(* Logix 5000 project; controller DUNEW2PLC1 vendor 1 type 14 code 221 rev 33.11; software revision 33.00; part 2 of 7 *)
(* tags used below, declared in another part *)
   AbortActive : BOOL;
   BOOLS : BOOL[1024];
   CheckCurSeg : BOOL;
   CheckNextSeg : BOOL;
   CmdA_Accel : REAL;
   CmdA_CircleType : DINT;
   CmdA_Decel : REAL;
   CmdA_Direction : DINT;
   CmdA_JerkAccel : REAL;
   CmdA_JerkDecel : REAL;
   CmdA_SegType : DINT;
   CmdA_Speed : REAL;
   CmdA_TermType : SINT;
   CmdA_ViaCenter : REAL[2];
   CmdA_XY : REAL[2];
   CmdB_Accel : REAL;
   CmdB_CircleType : DINT;
   CmdB_Decel : REAL;
   CmdB_Direction : DINT;
   CmdB_JerkAccel : REAL;
   CmdB_JerkDecel : REAL;
   CmdB_SegType : DINT;
   CmdB_Speed : REAL;
   CmdB_TermType : SINT;
   CmdB_ViaCenter : REAL[2];
   CmdB_XY : REAL[2];
   CmdTolerance : DINT;
   CurSeg : MotionSeg;
   DINTS : DINT[1024];
   EnqueueReq : BOOL;
   FaultCode : DINT;
   idx_0 : DINT;
   idx_2 : DINT;
   idx_3 : DINT;
   IssueCurPulse : BOOL;
   LoadCurReq : BOOL;
   MoveA : MOTION_INSTRUCTION;
   MoveB : MOTION_INSTRUCTION;
   NextSeg : MotionSeg;
   PrepCurMove : BOOL;
   PrepNextMove : BOOL;
   QueueCtl : CONTROL;
   QueueEmpty : BOOL;
   QueueStopReqONS : BOOL;
   REALS : REAL[1024];
   SegValid : BOOL;
   SegValidArc : BOOL;
   SegValidLine : BOOL;
   StartCurONS : BOOL;
   UseAasCurrent : BOOL;
   WaitCurAxisOn : BOOL;
   x_axis_mso : MOTION_INSTRUCTION;
   y_axis_mso : MOTION_INSTRUCTION;
   AbortQueue : BOOL;
   ActiveSeq : DINT;
   ALL_EOT_GOOD : BOOL;
   APA_IS_VERTICAL : BOOL;
   CurIssued : BOOL;
   ERROR_CODE : DINT;
   gui_stop : MOTION_INSTRUCTION;
   IncomingSeg : MotionSeg;
   IncomingSegAck : DINT;
   IncomingSegReqID : DINT;
   LastIncomingSegReqID : DINT;
   MAX_TOLERABLE_Z : REAL;
   MotionFault : BOOL;
   MOVE_TYPE : INT;   // 0 = No Move 1 = XY JOG 2 = XY Plane Move 3 = Z JOG 4 = Z Axis Move 5 = Toggle Latch Actuator 6 = Home the Latch Actuator
   NextIssued : BOOL;
   NEXTSTATE : DINT;
   QueueCount : DINT;
   QueueFault : BOOL;
   QueueFull : BOOL;
   QueueStopRequest : BOOL;
   SegQueue : MotionSeg[32];
   StartQueuedPath : BOOL;
   v_x_max : DINT;
   v_y_max : DINT;
   X_axis : AXIS_CIP_DRIVE;
   X_Y : COORDINATE_SYSTEM;
   Y_axis : AXIS_CIP_DRIVE;
   Z_axis : AXIS_CIP_DRIVE;
   Z_RETRACTED : BOOL;
(* queued_motion, continued *)

ROUTINE CapSegSpeed   (* ladder *)
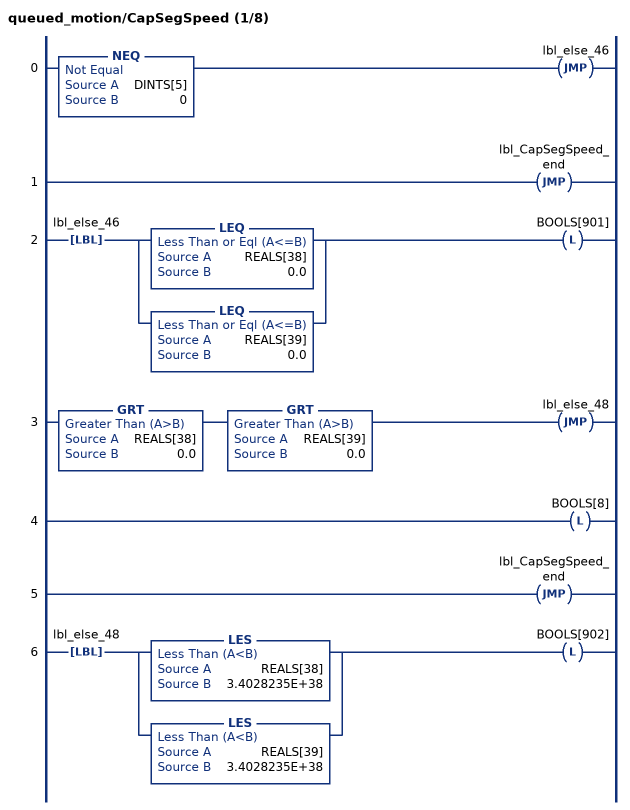
   0: NEQ(DINTS[5],0)JMP(lbl_else_46);
   1: JMP(lbl_CapSegSpeed_end);
   2: LBL(lbl_else_46)[LEQ(REALS[38],0.0) ,LEQ(REALS[39],0.0) ]OTL(BOOLS[901]);
   3: GRT(REALS[38],0.0)GRT(REALS[39],0.0)JMP(lbl_else_48);
   4: OTL(BOOLS[8]);
   5: JMP(lbl_CapSegSpeed_end);
   6: LBL(lbl_else_48)[LES(REALS[38],3.4028235E+38) ,LES(REALS[39],3.4028235E+38) ]OTL(BOOLS[902]);
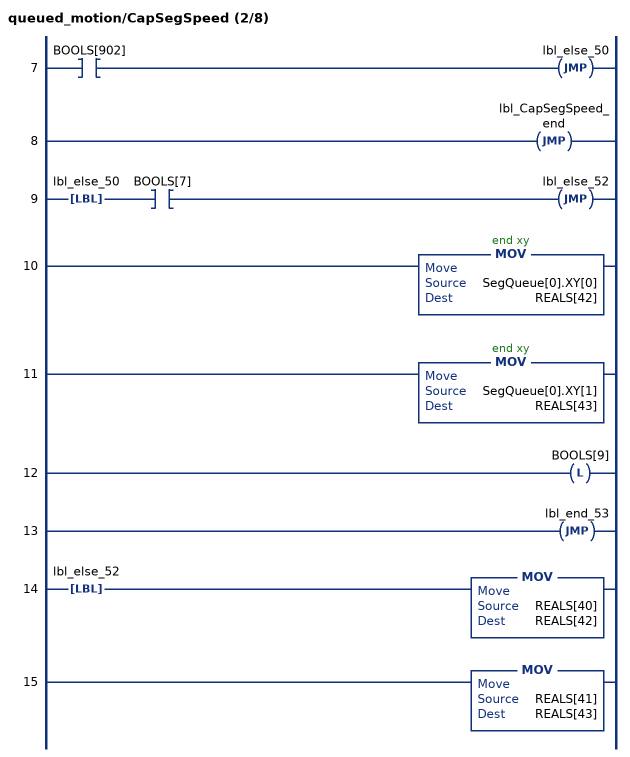
   7: XIC(BOOLS[902])JMP(lbl_else_50);
   8: JMP(lbl_CapSegSpeed_end);
   9: LBL(lbl_else_50)XIC(BOOLS[7])JMP(lbl_else_52);
   10: MOV(SegQueue[0].XY[0],REALS[42]);
   11: MOV(SegQueue[0].XY[1],REALS[43]);
   12: OTL(BOOLS[9]);
   13: JMP(lbl_end_53);
   14: LBL(lbl_else_52)MOV(REALS[40],REALS[42]);
   15: MOV(REALS[41],REALS[43]);
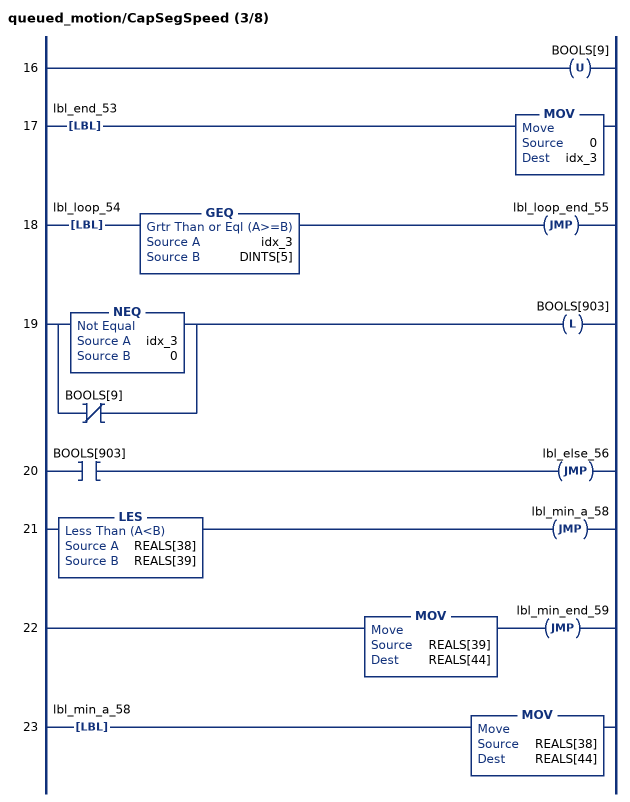
   16: OTU(BOOLS[9]);
   17: LBL(lbl_end_53)MOV(0,idx_3);
   18: LBL(lbl_loop_54)GEQ(idx_3,DINTS[5])JMP(lbl_loop_end_55);
   19: [NEQ(idx_3,0) ,XIO(BOOLS[9]) ]OTL(BOOLS[903]);
   20: XIC(BOOLS[903])JMP(lbl_else_56);
   21: LES(REALS[38],REALS[39])JMP(lbl_min_a_58);
   22: MOV(REALS[39],REALS[44])JMP(lbl_min_end_59);
   23: LBL(lbl_min_a_58)MOV(REALS[38],REALS[44]);
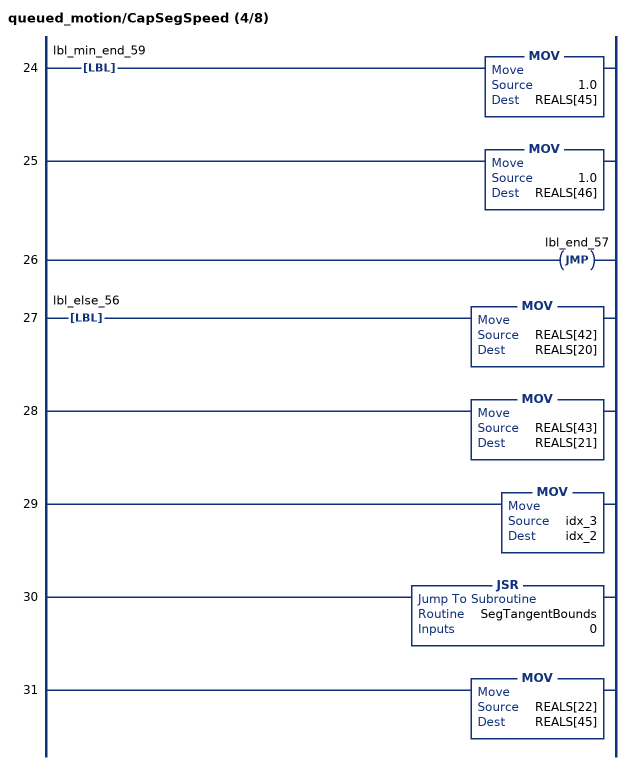
   24: LBL(lbl_min_end_59)MOV(1.0,REALS[45]);
   25: MOV(1.0,REALS[46]);
   26: JMP(lbl_end_57);
   27: LBL(lbl_else_56)MOV(REALS[42],REALS[20]);
   28: MOV(REALS[43],REALS[21]);
   29: MOV(idx_3,idx_2);
   30: JSR(SegTangentBounds,0);
   31: MOV(REALS[22],REALS[45]);
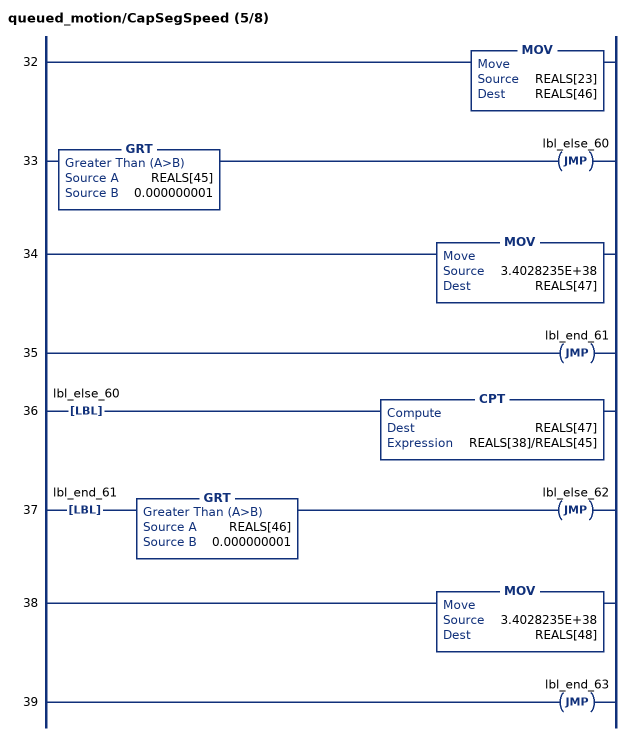
   32: MOV(REALS[23],REALS[46]);
   33: GRT(REALS[45],0.000000001)JMP(lbl_else_60);
   34: MOV(3.4028235E+38,REALS[47]);
   35: JMP(lbl_end_61);
   36: LBL(lbl_else_60)CPT(REALS[47],REALS[38]/REALS[45]);
   37: LBL(lbl_end_61)GRT(REALS[46],0.000000001)JMP(lbl_else_62);
   38: MOV(3.4028235E+38,REALS[48]);
   39: JMP(lbl_end_63);
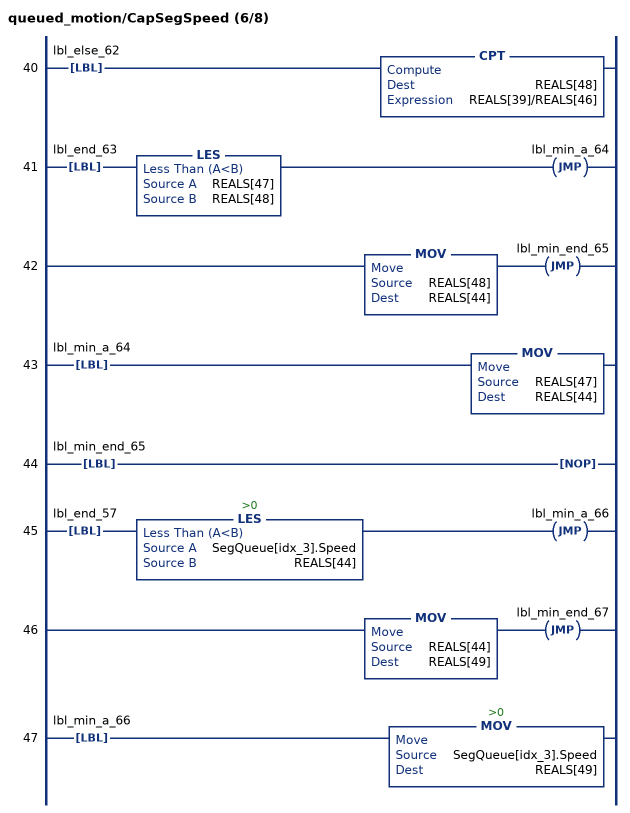
   40: LBL(lbl_else_62)CPT(REALS[48],REALS[39]/REALS[46]);
   41: LBL(lbl_end_63)LES(REALS[47],REALS[48])JMP(lbl_min_a_64);
   42: MOV(REALS[48],REALS[44])JMP(lbl_min_end_65);
   43: LBL(lbl_min_a_64)MOV(REALS[47],REALS[44]);
   44: LBL(lbl_min_end_65)NOP();
   45: LBL(lbl_end_57)LES(SegQueue[idx_3].Speed,REALS[44])JMP(lbl_min_a_66);
   46: MOV(REALS[44],REALS[49])JMP(lbl_min_end_67);
   47: LBL(lbl_min_a_66)MOV(SegQueue[idx_3].Speed,REALS[49]);
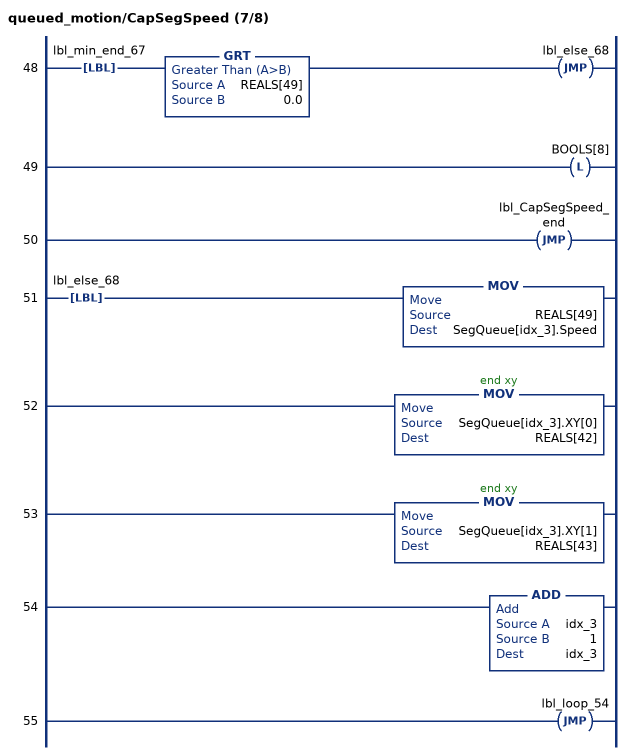
   48: LBL(lbl_min_end_67)GRT(REALS[49],0.0)JMP(lbl_else_68);
   49: OTL(BOOLS[8]);
   50: JMP(lbl_CapSegSpeed_end);
   51: LBL(lbl_else_68)MOV(REALS[49],SegQueue[idx_3].Speed);
   52: MOV(SegQueue[idx_3].XY[0],REALS[42]);
   53: MOV(SegQueue[idx_3].XY[1],REALS[43]);
   54: ADD(idx_3,1,idx_3);
   55: JMP(lbl_loop_54);
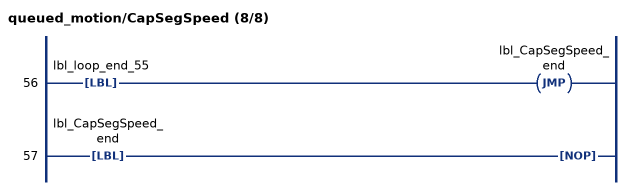
   56: LBL(lbl_loop_end_55)JMP(lbl_CapSegSpeed_end);
   57: LBL(lbl_CapSegSpeed_end)NOP();
END_ROUTINE

ROUTINE CircleCenterForSeg   (* ladder *)
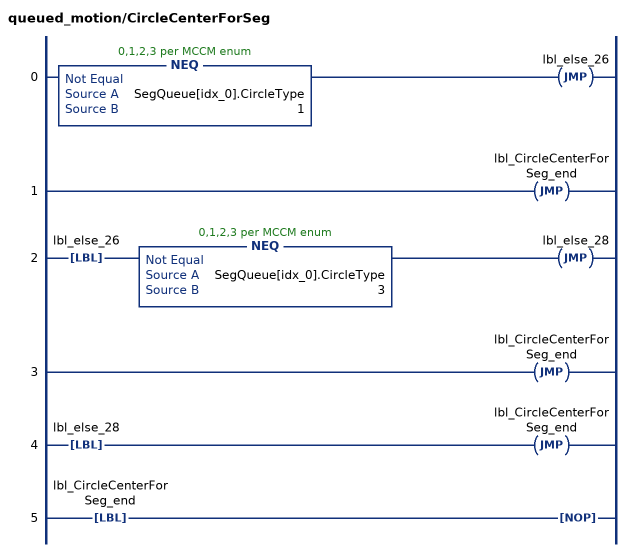
   0: NEQ(SegQueue[idx_0].CircleType,1)JMP(lbl_else_26);
   1: JMP(lbl_CircleCenterForSeg_end);
   2: LBL(lbl_else_26)NEQ(SegQueue[idx_0].CircleType,3)JMP(lbl_else_28);
   3: JMP(lbl_CircleCenterForSeg_end);
   4: LBL(lbl_else_28)JMP(lbl_CircleCenterForSeg_end);
   5: LBL(lbl_CircleCenterForSeg_end)NOP();
END_ROUTINE

ROUTINE main   (* ladder *)
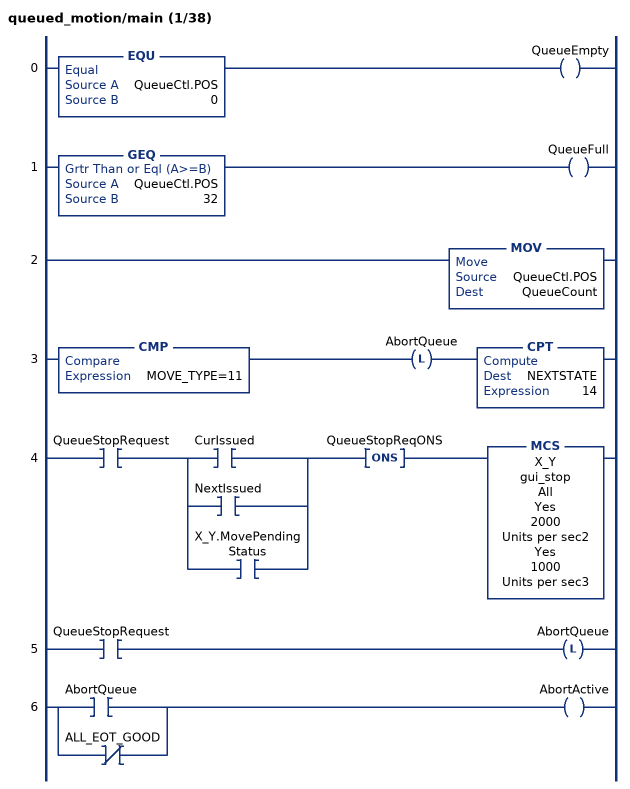
   0: EQU(QueueCtl.POS,0)OTE(QueueEmpty);
   1: GEQ(QueueCtl.POS,32)OTE(QueueFull);
   2: MOV(QueueCtl.POS,QueueCount);
   3: CMP(MOVE_TYPE=11)OTL(AbortQueue)CPT(NEXTSTATE,14);
   4: XIC(QueueStopRequest)[XIC(CurIssued) ,XIC(NextIssued) ,XIC(X_Y.MovePendingStatus) ]ONS(QueueStopReqONS)MCS(X_Y,gui_stop,All,Yes,2000,Units per sec2,Yes,1000,Units per sec3);
   5: XIC(QueueStopRequest)OTL(AbortQueue);
   6: [XIC(AbortQueue) ,XIO(ALL_EOT_GOOD) ]OTE(AbortActive);
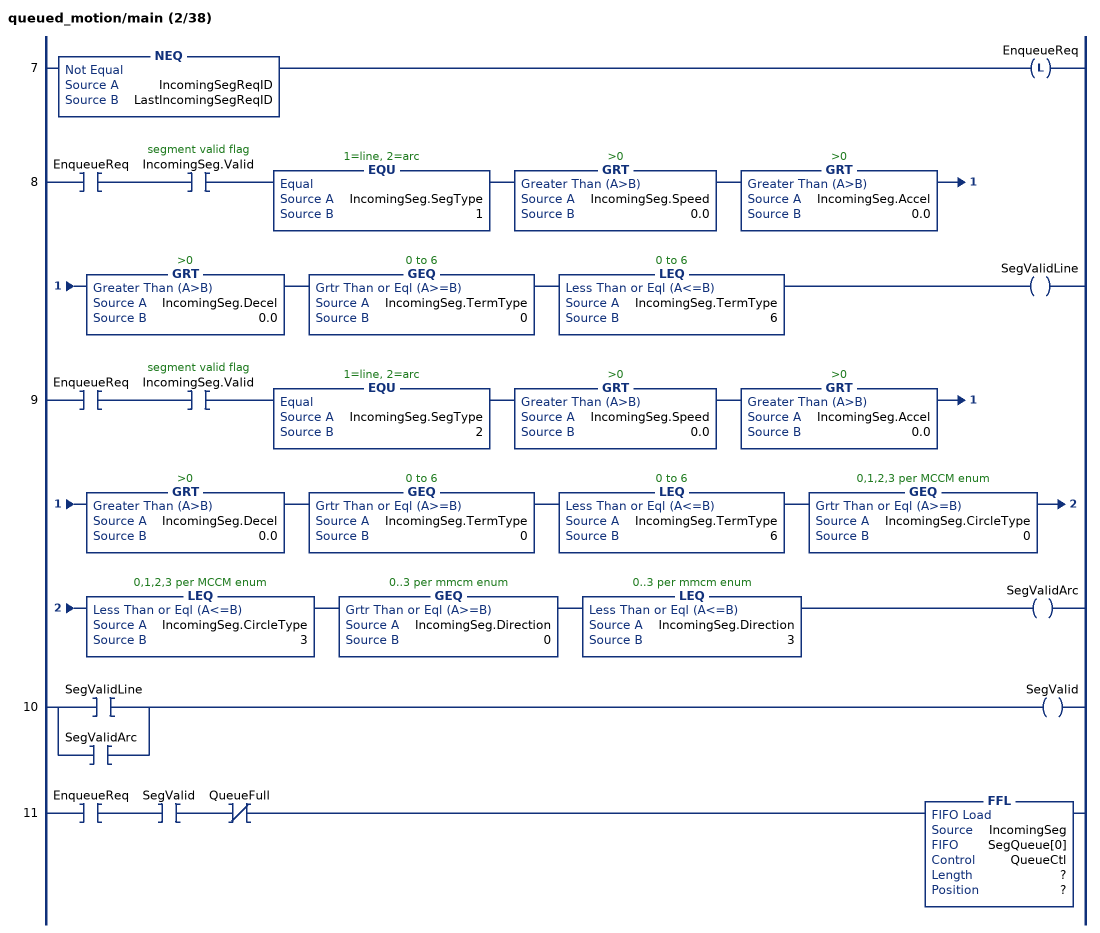
   7: NEQ(IncomingSegReqID,LastIncomingSegReqID)OTL(EnqueueReq);
   8: XIC(EnqueueReq)XIC(IncomingSeg.Valid)EQU(IncomingSeg.SegType,1)GRT(IncomingSeg.Speed,0.0)GRT(IncomingSeg.Accel,0.0)GRT(IncomingSeg.Decel,0.0)GEQ(IncomingSeg.TermType,0)LEQ(IncomingSeg.TermType,6)OTE(SegValidLine);
   9: XIC(EnqueueReq)XIC(IncomingSeg.Valid)EQU(IncomingSeg.SegType,2)GRT(IncomingSeg.Speed,0.0)GRT(IncomingSeg.Accel,0.0)GRT(IncomingSeg.Decel,0.0)GEQ(IncomingSeg.TermType,0)LEQ(IncomingSeg.TermType,6)GEQ(IncomingSeg.CircleType,0)LEQ(IncomingSeg.CircleType,3)GEQ(IncomingSeg.Direction,0)LEQ(IncomingSeg.Direction,3)OTE(SegValidArc);
   10: [XIC(SegValidLine) ,XIC(SegValidArc) ]OTE(SegValid);
   11: XIC(EnqueueReq)XIC(SegValid)XIO(QueueFull)FFL(IncomingSeg,SegQueue[0],QueueCtl,?,?);
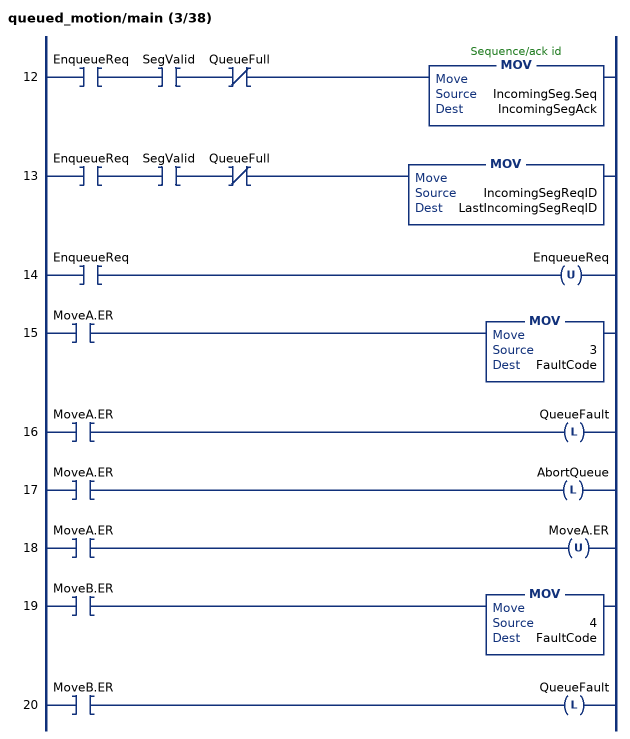
   12: XIC(EnqueueReq)XIC(SegValid)XIO(QueueFull)MOV(IncomingSeg.Seq,IncomingSegAck);
   13: XIC(EnqueueReq)XIC(SegValid)XIO(QueueFull)MOV(IncomingSegReqID,LastIncomingSegReqID);
   14: XIC(EnqueueReq)OTU(EnqueueReq);
   15: XIC(MoveA.ER)MOV(3,FaultCode);
   16: XIC(MoveA.ER)OTL(QueueFault);
   17: XIC(MoveA.ER)OTL(AbortQueue);
   18: XIC(MoveA.ER)OTU(MoveA.ER);
   19: XIC(MoveB.ER)MOV(4,FaultCode);
   20: XIC(MoveB.ER)OTL(QueueFault);
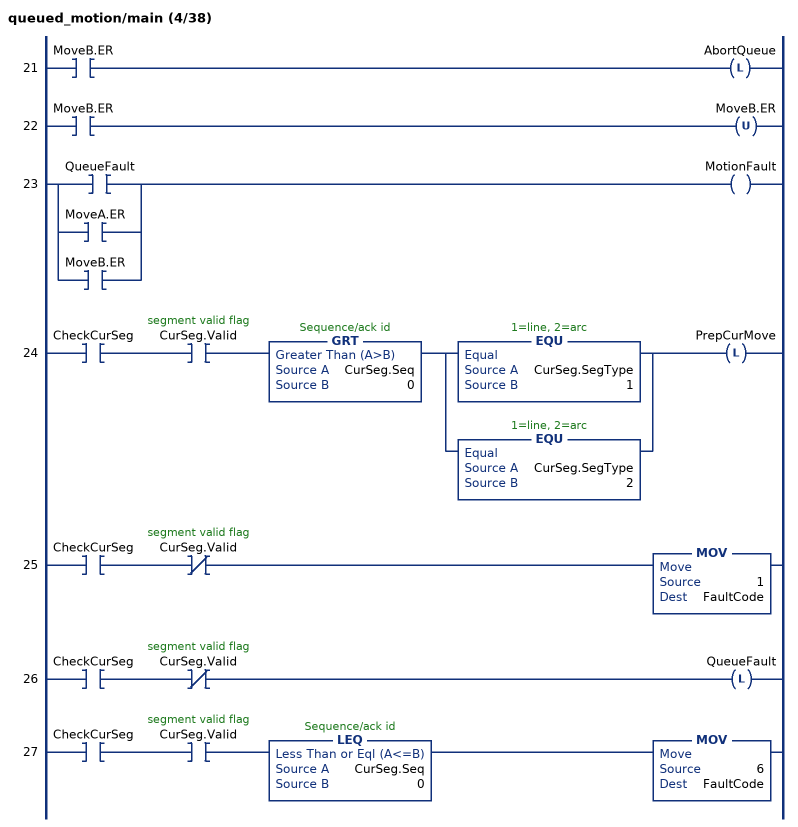
   21: XIC(MoveB.ER)OTL(AbortQueue);
   22: XIC(MoveB.ER)OTU(MoveB.ER);
   23: [XIC(QueueFault) ,XIC(MoveA.ER) ,XIC(MoveB.ER) ]OTE(MotionFault);
   24: XIC(CheckCurSeg)XIC(CurSeg.Valid)GRT(CurSeg.Seq,0)[EQU(CurSeg.SegType,1) ,EQU(CurSeg.SegType,2) ]OTL(PrepCurMove);
   25: XIC(CheckCurSeg)XIO(CurSeg.Valid)MOV(1,FaultCode);
   26: XIC(CheckCurSeg)XIO(CurSeg.Valid)OTL(QueueFault);
   27: XIC(CheckCurSeg)XIC(CurSeg.Valid)LEQ(CurSeg.Seq,0)MOV(6,FaultCode);
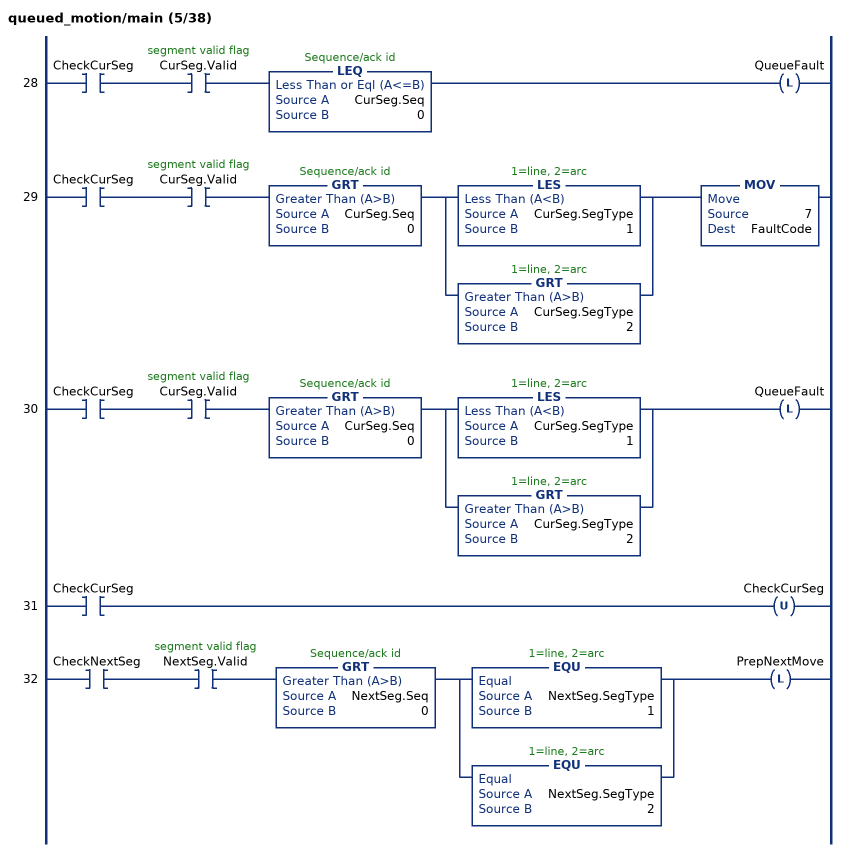
   28: XIC(CheckCurSeg)XIC(CurSeg.Valid)LEQ(CurSeg.Seq,0)OTL(QueueFault);
   29: XIC(CheckCurSeg)XIC(CurSeg.Valid)GRT(CurSeg.Seq,0)[LES(CurSeg.SegType,1) ,GRT(CurSeg.SegType,2) ]MOV(7,FaultCode);
   30: XIC(CheckCurSeg)XIC(CurSeg.Valid)GRT(CurSeg.Seq,0)[LES(CurSeg.SegType,1) ,GRT(CurSeg.SegType,2) ]OTL(QueueFault);
   31: XIC(CheckCurSeg)OTU(CheckCurSeg);
   32: XIC(CheckNextSeg)XIC(NextSeg.Valid)GRT(NextSeg.Seq,0)[EQU(NextSeg.SegType,1) ,EQU(NextSeg.SegType,2) ]OTL(PrepNextMove);
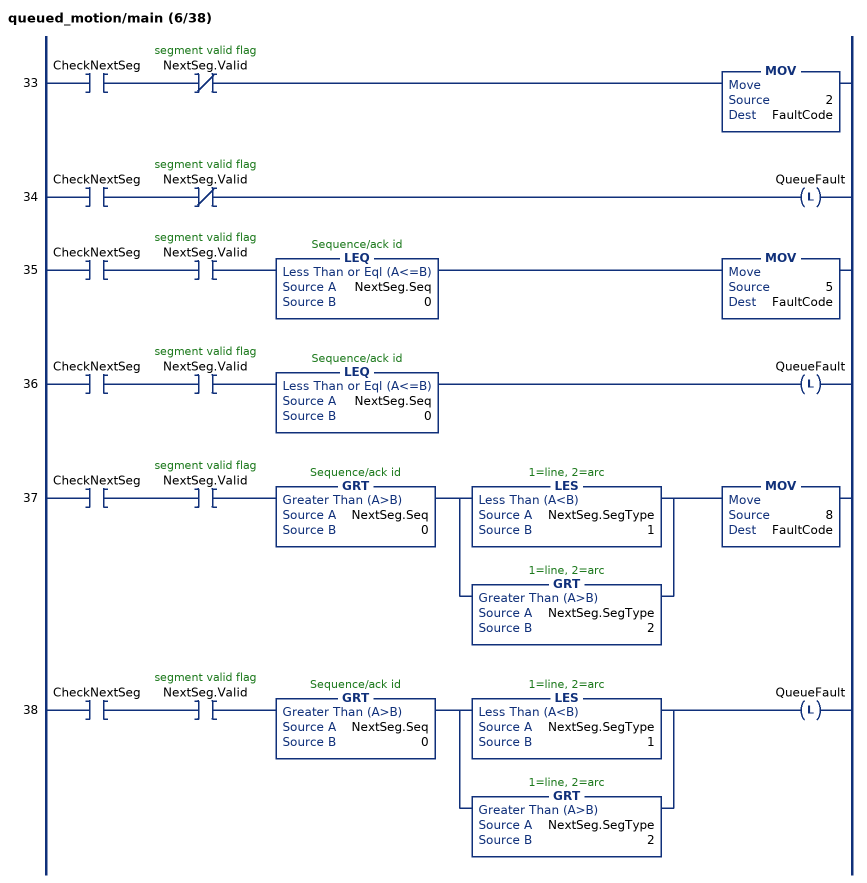
   33: XIC(CheckNextSeg)XIO(NextSeg.Valid)MOV(2,FaultCode);
   34: XIC(CheckNextSeg)XIO(NextSeg.Valid)OTL(QueueFault);
   35: XIC(CheckNextSeg)XIC(NextSeg.Valid)LEQ(NextSeg.Seq,0)MOV(5,FaultCode);
   36: XIC(CheckNextSeg)XIC(NextSeg.Valid)LEQ(NextSeg.Seq,0)OTL(QueueFault);
   37: XIC(CheckNextSeg)XIC(NextSeg.Valid)GRT(NextSeg.Seq,0)[LES(NextSeg.SegType,1) ,GRT(NextSeg.SegType,2) ]MOV(8,FaultCode);
   38: XIC(CheckNextSeg)XIC(NextSeg.Valid)GRT(NextSeg.Seq,0)[LES(NextSeg.SegType,1) ,GRT(NextSeg.SegType,2) ]OTL(QueueFault);
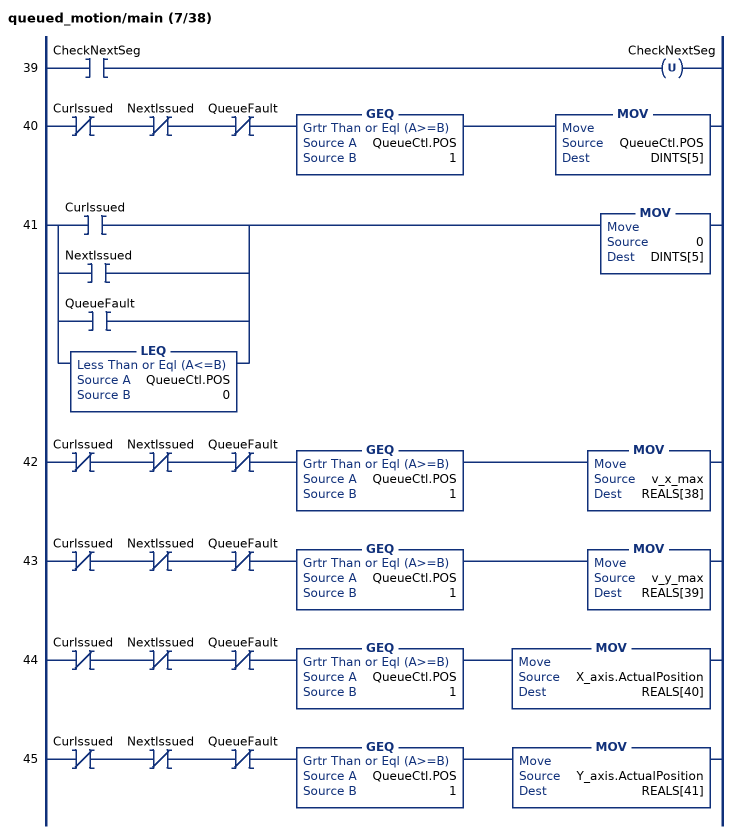
   39: XIC(CheckNextSeg)OTU(CheckNextSeg);
   40: XIO(CurIssued)XIO(NextIssued)XIO(QueueFault)GEQ(QueueCtl.POS,1)MOV(QueueCtl.POS,DINTS[5]);
   41: [XIC(CurIssued) ,XIC(NextIssued) ,XIC(QueueFault) ,LEQ(QueueCtl.POS,0) ]MOV(0,DINTS[5]);
   42: XIO(CurIssued)XIO(NextIssued)XIO(QueueFault)GEQ(QueueCtl.POS,1)MOV(v_x_max,REALS[38]);
   43: XIO(CurIssued)XIO(NextIssued)XIO(QueueFault)GEQ(QueueCtl.POS,1)MOV(v_y_max,REALS[39]);
   44: XIO(CurIssued)XIO(NextIssued)XIO(QueueFault)GEQ(QueueCtl.POS,1)MOV(X_axis.ActualPosition,REALS[40]);
   45: XIO(CurIssued)XIO(NextIssued)XIO(QueueFault)GEQ(QueueCtl.POS,1)MOV(Y_axis.ActualPosition,REALS[41]);
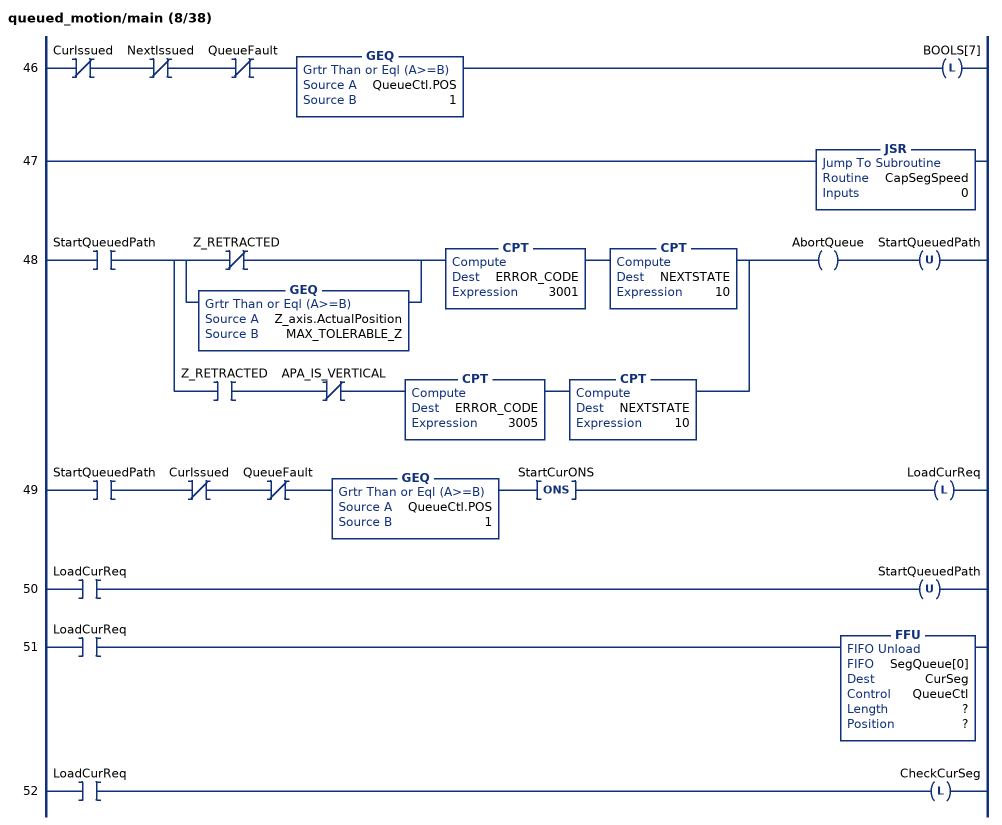
   46: XIO(CurIssued)XIO(NextIssued)XIO(QueueFault)GEQ(QueueCtl.POS,1)OTL(BOOLS[7]);
   47: JSR(CapSegSpeed,0);
   48: XIC(StartQueuedPath)[[XIO(Z_RETRACTED) ,GEQ(Z_axis.ActualPosition,MAX_TOLERABLE_Z) ] CPT(ERROR_CODE,3001) CPT(NEXTSTATE,10) ,XIC(Z_RETRACTED) XIO(APA_IS_VERTICAL) CPT(ERROR_CODE,3005) CPT(NEXTSTATE,10) ]OTE(AbortQueue)OTU(StartQueuedPath);
   49: XIC(StartQueuedPath)XIO(CurIssued)XIO(QueueFault)GEQ(QueueCtl.POS,1)ONS(StartCurONS)OTL(LoadCurReq);
   50: XIC(LoadCurReq)OTU(StartQueuedPath);
   51: XIC(LoadCurReq)FFU(SegQueue[0],CurSeg,QueueCtl,?,?);
   52: XIC(LoadCurReq)OTL(CheckCurSeg);
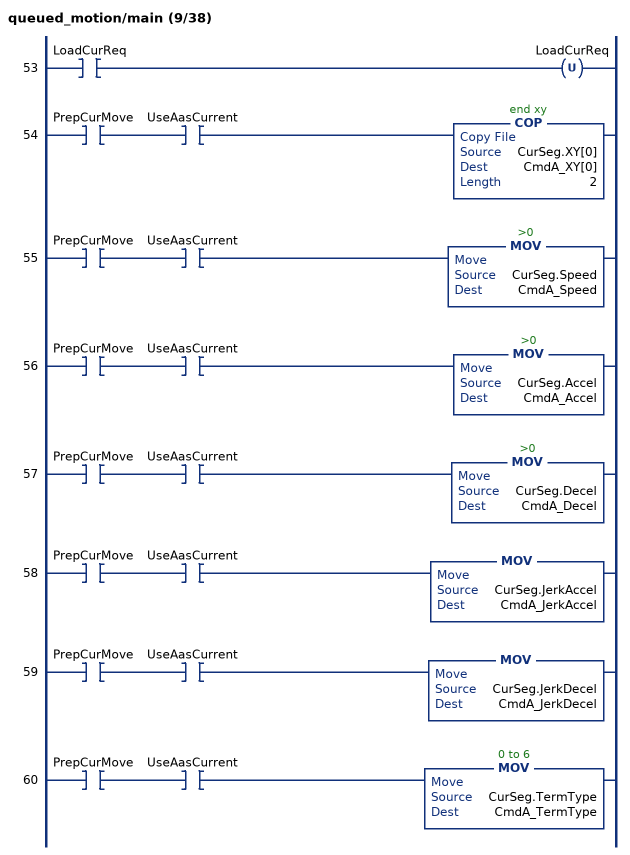
   53: XIC(LoadCurReq)OTU(LoadCurReq);
   54: XIC(PrepCurMove)XIC(UseAasCurrent)COP(CurSeg.XY[0],CmdA_XY[0],2);
   55: XIC(PrepCurMove)XIC(UseAasCurrent)MOV(CurSeg.Speed,CmdA_Speed);
   56: XIC(PrepCurMove)XIC(UseAasCurrent)MOV(CurSeg.Accel,CmdA_Accel);
   57: XIC(PrepCurMove)XIC(UseAasCurrent)MOV(CurSeg.Decel,CmdA_Decel);
   58: XIC(PrepCurMove)XIC(UseAasCurrent)MOV(CurSeg.JerkAccel,CmdA_JerkAccel);
   59: XIC(PrepCurMove)XIC(UseAasCurrent)MOV(CurSeg.JerkDecel,CmdA_JerkDecel);
   60: XIC(PrepCurMove)XIC(UseAasCurrent)MOV(CurSeg.TermType,CmdA_TermType);
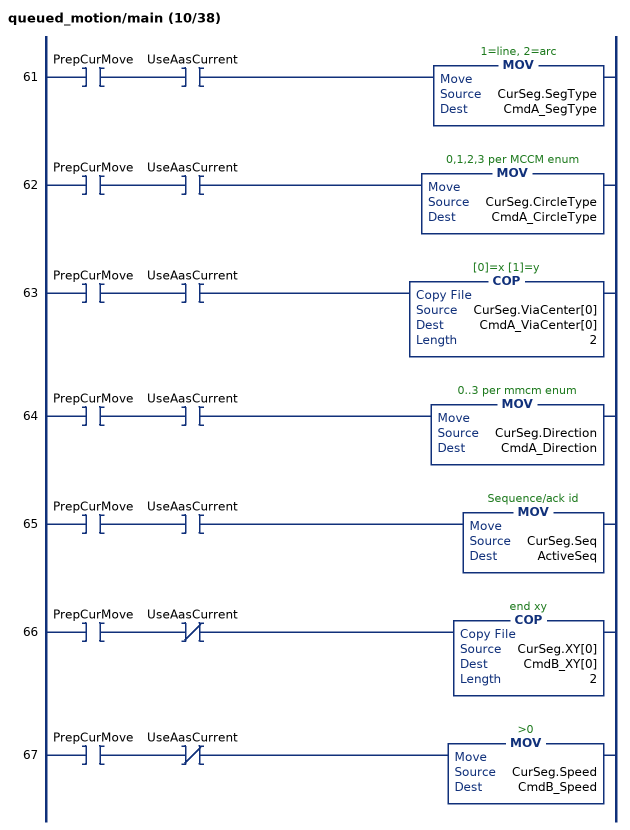
   61: XIC(PrepCurMove)XIC(UseAasCurrent)MOV(CurSeg.SegType,CmdA_SegType);
   62: XIC(PrepCurMove)XIC(UseAasCurrent)MOV(CurSeg.CircleType,CmdA_CircleType);
   63: XIC(PrepCurMove)XIC(UseAasCurrent)COP(CurSeg.ViaCenter[0],CmdA_ViaCenter[0],2);
   64: XIC(PrepCurMove)XIC(UseAasCurrent)MOV(CurSeg.Direction,CmdA_Direction);
   65: XIC(PrepCurMove)XIC(UseAasCurrent)MOV(CurSeg.Seq,ActiveSeq);
   66: XIC(PrepCurMove)XIO(UseAasCurrent)COP(CurSeg.XY[0],CmdB_XY[0],2);
   67: XIC(PrepCurMove)XIO(UseAasCurrent)MOV(CurSeg.Speed,CmdB_Speed);
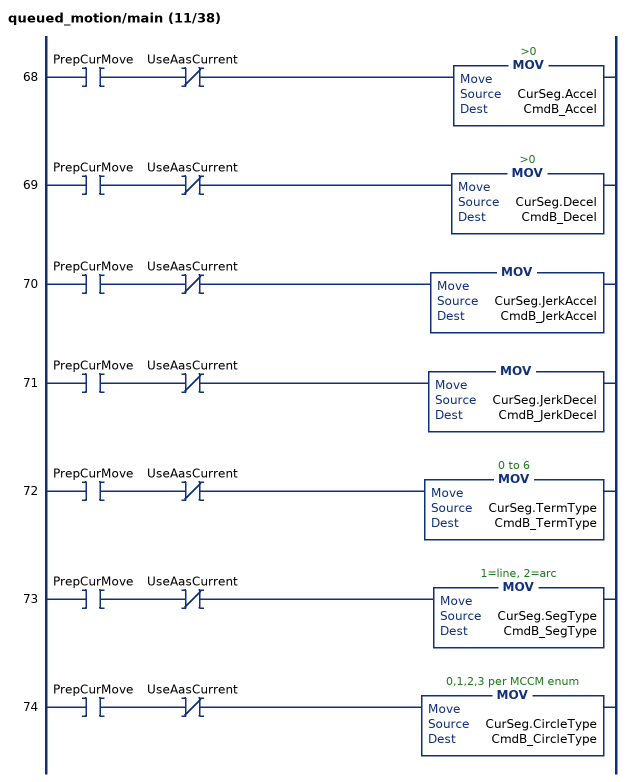
   68: XIC(PrepCurMove)XIO(UseAasCurrent)MOV(CurSeg.Accel,CmdB_Accel);
   69: XIC(PrepCurMove)XIO(UseAasCurrent)MOV(CurSeg.Decel,CmdB_Decel);
   70: XIC(PrepCurMove)XIO(UseAasCurrent)MOV(CurSeg.JerkAccel,CmdB_JerkAccel);
   71: XIC(PrepCurMove)XIO(UseAasCurrent)MOV(CurSeg.JerkDecel,CmdB_JerkDecel);
   72: XIC(PrepCurMove)XIO(UseAasCurrent)MOV(CurSeg.TermType,CmdB_TermType);
   73: XIC(PrepCurMove)XIO(UseAasCurrent)MOV(CurSeg.SegType,CmdB_SegType);
   74: XIC(PrepCurMove)XIO(UseAasCurrent)MOV(CurSeg.CircleType,CmdB_CircleType);
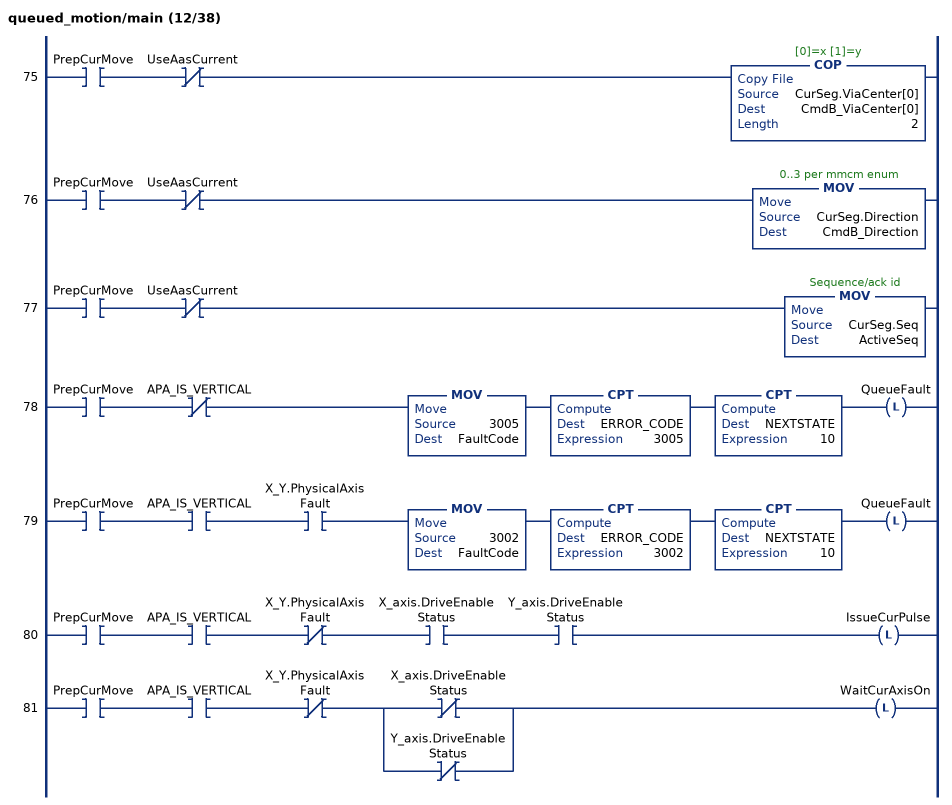
   75: XIC(PrepCurMove)XIO(UseAasCurrent)COP(CurSeg.ViaCenter[0],CmdB_ViaCenter[0],2);
   76: XIC(PrepCurMove)XIO(UseAasCurrent)MOV(CurSeg.Direction,CmdB_Direction);
   77: XIC(PrepCurMove)XIO(UseAasCurrent)MOV(CurSeg.Seq,ActiveSeq);
   78: XIC(PrepCurMove)XIO(APA_IS_VERTICAL)MOV(3005,FaultCode)CPT(ERROR_CODE,3005)CPT(NEXTSTATE,10)OTL(QueueFault);
   79: XIC(PrepCurMove)XIC(APA_IS_VERTICAL)XIC(X_Y.PhysicalAxisFault)MOV(3002,FaultCode)CPT(ERROR_CODE,3002)CPT(NEXTSTATE,10)OTL(QueueFault);
   80: XIC(PrepCurMove)XIC(APA_IS_VERTICAL)XIO(X_Y.PhysicalAxisFault)XIC(X_axis.DriveEnableStatus)XIC(Y_axis.DriveEnableStatus)OTL(IssueCurPulse);
   81: XIC(PrepCurMove)XIC(APA_IS_VERTICAL)XIO(X_Y.PhysicalAxisFault)[XIO(X_axis.DriveEnableStatus) ,XIO(Y_axis.DriveEnableStatus) ]OTL(WaitCurAxisOn);
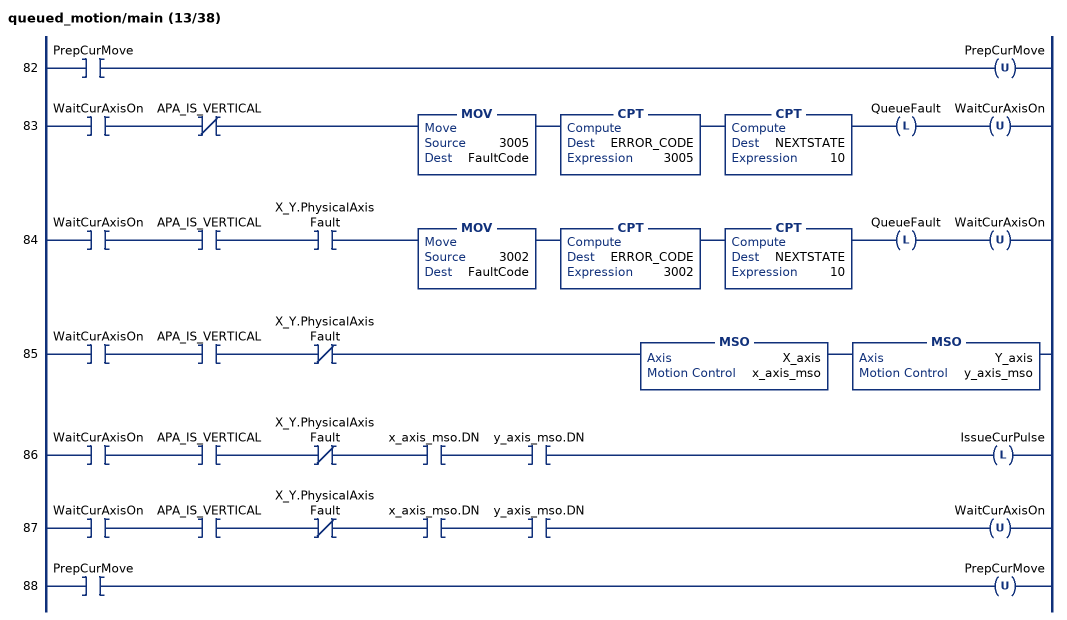
   82: XIC(PrepCurMove)OTU(PrepCurMove);
   83: XIC(WaitCurAxisOn)XIO(APA_IS_VERTICAL)MOV(3005,FaultCode)CPT(ERROR_CODE,3005)CPT(NEXTSTATE,10)OTL(QueueFault)OTU(WaitCurAxisOn);
   84: XIC(WaitCurAxisOn)XIC(APA_IS_VERTICAL)XIC(X_Y.PhysicalAxisFault)MOV(3002,FaultCode)CPT(ERROR_CODE,3002)CPT(NEXTSTATE,10)OTL(QueueFault)OTU(WaitCurAxisOn);
   85: XIC(WaitCurAxisOn)XIC(APA_IS_VERTICAL)XIO(X_Y.PhysicalAxisFault)MSO(X_axis,x_axis_mso)MSO(Y_axis,y_axis_mso);
   86: XIC(WaitCurAxisOn)XIC(APA_IS_VERTICAL)XIO(X_Y.PhysicalAxisFault)XIC(x_axis_mso.DN)XIC(y_axis_mso.DN)OTL(IssueCurPulse);
   87: XIC(WaitCurAxisOn)XIC(APA_IS_VERTICAL)XIO(X_Y.PhysicalAxisFault)XIC(x_axis_mso.DN)XIC(y_axis_mso.DN)OTU(WaitCurAxisOn);
   88: XIC(PrepCurMove)OTU(PrepCurMove);
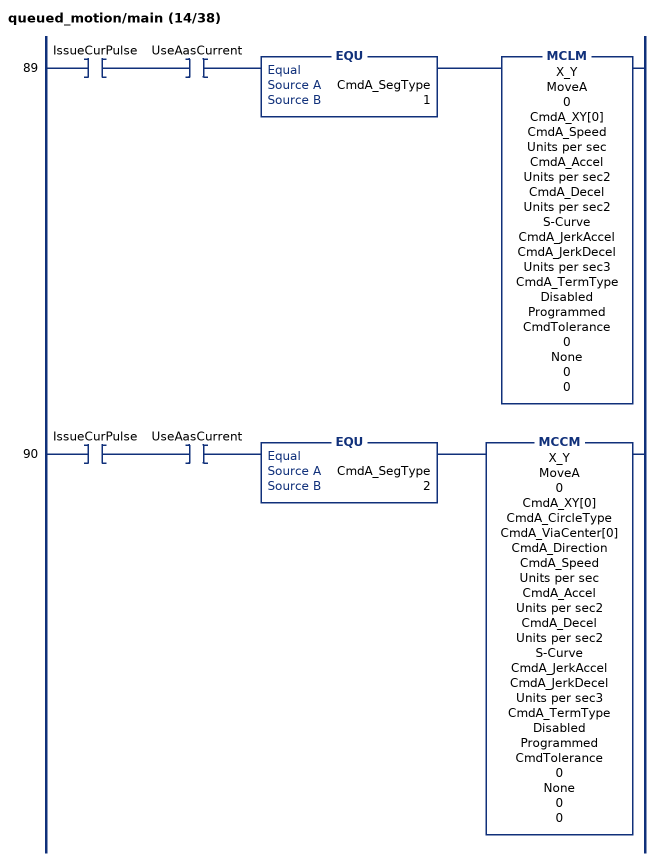
   89: XIC(IssueCurPulse)XIC(UseAasCurrent)EQU(CmdA_SegType,1)MCLM(X_Y,MoveA,0,CmdA_XY[0],CmdA_Speed,Units per sec,CmdA_Accel,Units per sec2,CmdA_Decel,Units per sec2,S-Curve,CmdA_JerkAccel,CmdA_JerkDecel,Units per sec3,CmdA_TermType,Disabled,Programmed,CmdTolerance,0,None,0,0);
   90: XIC(IssueCurPulse)XIC(UseAasCurrent)EQU(CmdA_SegType,2)MCCM(X_Y,MoveA,0,CmdA_XY[0],CmdA_CircleType,CmdA_ViaCenter[0],CmdA_Direction,CmdA_Speed,Units per sec,CmdA_Accel,Units per sec2,CmdA_Decel,Units per sec2,S-Curve,CmdA_JerkAccel,CmdA_JerkDecel,Units per sec3,CmdA_TermType,Disabled,Programmed,CmdTolerance,0,None,0,0);
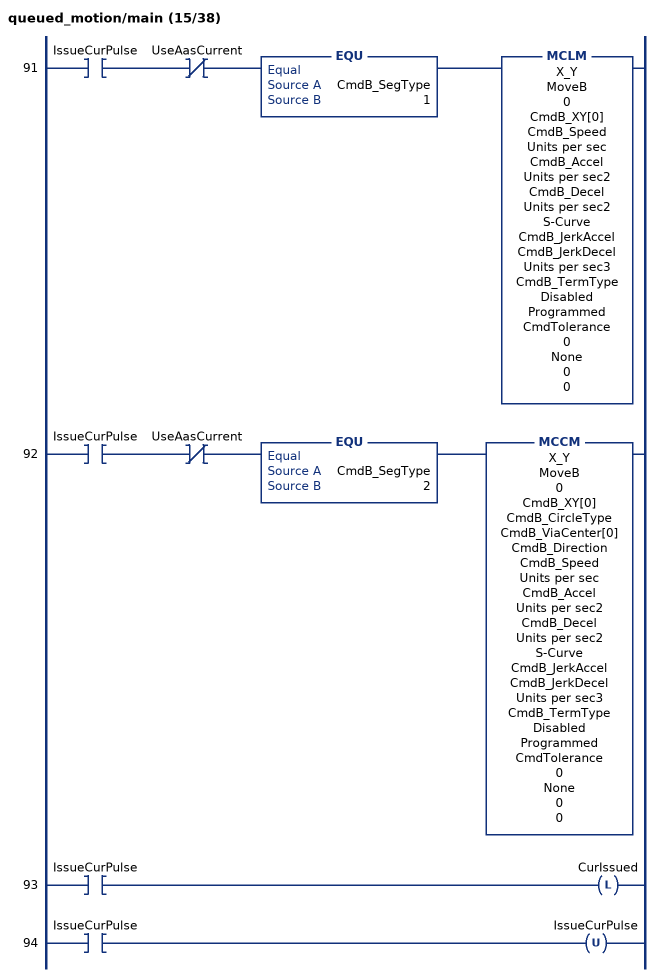
   91: XIC(IssueCurPulse)XIO(UseAasCurrent)EQU(CmdB_SegType,1)MCLM(X_Y,MoveB,0,CmdB_XY[0],CmdB_Speed,Units per sec,CmdB_Accel,Units per sec2,CmdB_Decel,Units per sec2,S-Curve,CmdB_JerkAccel,CmdB_JerkDecel,Units per sec3,CmdB_TermType,Disabled,Programmed,CmdTolerance,0,None,0,0);
   92: XIC(IssueCurPulse)XIO(UseAasCurrent)EQU(CmdB_SegType,2)MCCM(X_Y,MoveB,0,CmdB_XY[0],CmdB_CircleType,CmdB_ViaCenter[0],CmdB_Direction,CmdB_Speed,Units per sec,CmdB_Accel,Units per sec2,CmdB_Decel,Units per sec2,S-Curve,CmdB_JerkAccel,CmdB_JerkDecel,Units per sec3,CmdB_TermType,Disabled,Programmed,CmdTolerance,0,None,0,0);
   93: XIC(IssueCurPulse)OTL(CurIssued);
   94: XIC(IssueCurPulse)OTU(IssueCurPulse);
